// TwinCAT 3 PLC project TwinCAT_OpenFramework_Collections
// Title: TwinCAT Open Framework Collections
// Company: Oleksandr Tiutyk FOP
// Author: Oleksandr Tiutyk
// ProjectVersion: 1.0.13.0
// Description: Dynamic and static collections for TwinCAT.OpenFramework: ByteList, List, Dictionary, UniqueDataSet, Queue, Stack
// ProgramVersion: 3.1.4026.28
// libraries:
//   Tc2_Standard, * (Beckhoff Automation GmbH)
//   Tc2_System, * (Beckhoff Automation GmbH)
//   [TwinCAT Open Framework Core], * (Oleksandr Tiutyk FOP)
// project tree:
//   ByteList/ ByteList.TcPOU, ByteListEnumerator.TcPOU, IByteList.TcIO, IReadOnlyByteList.TcIO
//   Dictionary/ Dictionary.TcPOU, DictionaryEnumerator.TcPOU, IDictionary.TcIO, IReadOnlyDictionary.TcIO
//   / ICollection.TcIO
//   Internal/ CurrentNamespace.TcPOU, NamespaceExtractor.TcPOU
//   List/ IList.TcIO, IReadOnlyList.TcIO, List.TcPOU, ListEnumerator.TcPOU (not stored)
//   Queue/ IReadOnlyQueue.TcIO, IQueue.TcIO, Queue.TcPOU (not stored), QueueEnumerator.TcPOU
//   Stack/ IReadOnlyStack.TcIO, IStack.TcIO, Stack.TcPOU, StackEnumerator.TcPOU
//   UniqueDataSet/ UniqueDataSet.TcPOU, UniqueDataSetEnumerator.TcPOU, IUniqueDataSet.TcIO, IReadOnlyUniqueDataSet.TcIO
//   Version/ Global_Version.TcGVL
// (motion and I/O tree: see PLC project twincat_openframework_core)
// real-time tasks:
//   TASK PlcTask: cycle T#10ms, priority 20, ADS port 350
//   TASK TestTask: cycle T#10ms, priority 1, ADS port 351
//   TASK RunnerTestTask: cycle T#10ms, priority 2, ADS port 354
//   TASK HowToTask: cycle T#10ms, priority 22, ADS port 353
// variable links:

// ---- Version/Global_Version.TcGVL
{attribute 'TcGenerated'}
{attribute 'no-analysis'}
{attribute 'linkalways'}
// This function has been automatically generated from the project information.
VAR_GLOBAL CONSTANT
	{attribute 'const_non_replaced'}
	stLibVersion_TwinCAT_Open_Framework_Collections : ST_LibVersion := (iMajor := 1, iMinor := 0, iBuild := 13, iRevision := 0, nFlags := 0, sVersion := '1.0.13.0');
END_VAR

// ---- ByteList/IByteList.TcIO
(*
SPDX-FileCopyrightText: © 2026 Oleksandr Tiutyk <trofimich@gmail.com>
SPDX-License-Identifier: MIT
License: https://opensource.org/license/mit
*)

(*!
<summary>Provides byte sequence mutation and raw-memory copying.</summary>
<description>
Append adds bytes. LoadFrom writes at startIndex and sets Length to the end of the copied range, potentially
truncating the old tail. Input memory is borrowed for copying, never adopted. Remove by value is a no-op when
the value is absent, including on an empty collection. See method declarations for current safety limitations.
</description>
*)

INTERFACE IByteList EXTENDS IReadOnlyByteList

(*!
<summary>Appends the raw storage bytes of an ANY argument.</summary>
<description>
Borrows the argument for copying and uses its full runtime size, including string capacity and structure
padding. Not portable serialization or object cloning. Shares AppendData capacity checks, overlap support and
failure behavior.
</description>
*)
METHOD AppendAny : IByteList
VAR_INPUT
	data : ANY;
END_VAR
END_METHOD

(*!
<summary>Appends one byte by value.</summary>
<description>
Returns this list. Full static storage raises an exception; dynamic growth uses checked allocation and
terminal OOM handling.
</description>
*)
METHOD AppendByte : IByteList
VAR_INPUT
	value : BYTE;
END_VAR
END_METHOD

(*!
<summary>Appends bytes copied from a borrowed memory range.</summary>
<description>
Null data or zero dataSize is a no-op before size validation. Otherwise the source must be readable and
negative sizes or a resulting length outside DINT raise ArgumentOutOfRangeException before copying. Static
capacity exhaustion raises StaticCollectionFullException. Dynamic allocation uses checked growth and terminal
OOM handling. The existing growth increment (free capacity plus input size) is retained and must also fit. The
source may refer to this collection buffer, including overlapping ranges. The caller must provide a readable
range of dataSize bytes; growth keeps the old buffer alive until copying completes. No restriction to logical
Length is imposed on the source. Returns this list.
</description>
*)
METHOD AppendData : IByteList
VAR_INPUT
	data : POINTER TO BYTE;
	dataSize : TOF_Core.DINT_LENGTH;
END_VAR
END_METHOD

(*!
<summary>Appends the raw bytes referenced by a generic descriptor.</summary>
<description>
Borrows the descriptor without adopting or releasing it. Copies Address and Size without value conversion or
object cloning. Size above SignedInt32.MAX_VALUE raises ArgumentOutOfRangeException before narrowing,
including for a null Address. Shares AppendData aliasing and failure behavior.
</description>
*)
METHOD AppendGeneric : IByteList
VAR_INPUT
	data : TOF_Core.GENERIC_VALUE;
END_VAR
END_METHOD

(*!
<summary>Resets the byte count and optionally releases dynamic storage.</summary>
<description>
The default retains capacity for reuse. releaseDynamicMemory = TRUE deletes dynamic storage and sets capacity
to zero. Static storage is retained. Returns this list; old contents are no longer logical entries.
</description>
*)
METHOD Clear : IByteList
VAR_INPUT
	releaseDynamicMemory : BOOL := FALSE;
END_VAR
END_METHOD

(*!
<summary>Loads the full raw representation of an ANY argument at a position.</summary>
<description>
Delegates to LoadFromData using the runtime byte size, including padding and string capacity. Borrows the
source and may truncate the previous tail. Shares LoadFromData limits; not portable serialization.
</description>
*)
METHOD LoadFromAny : IByteList
VAR_INPUT
	data : ANY;
	startIndex : TOF_Core.DINT_INDEX := 0;
END_VAR
END_METHOD

(*!
<summary>Copies bytes at a position and sets Length to the end of the copy.</summary>
<description>
startIndex must lie between zero and old Length inclusive, and dataSize must be nonnegative; invalid arguments
raise ArgumentOutOfRangeException. Null data or zero size leaves Length unchanged after these checks. For a
nonempty copy, the resulting length is checked against DINT before arithmetic or mutation. The prefix remains
and the tail beyond the new end is logically truncated. Static capacity exhaustion raises
StaticCollectionFullException; dynamic growth uses checked allocation and terminal OOM handling. Internal
sources and overlapping ranges are supported. The caller must provide a readable source range of dataSize
bytes; the old buffer remains alive throughout copying on growth. No restriction to logical Length is imposed
on the source. Returns this list.
</description>
*)
METHOD LoadFromData : IByteList
VAR_INPUT
	data : POINTER TO BYTE;
	dataSize : TOF_Core.DINT_LENGTH;
	startIndex : TOF_Core.DINT_INDEX := 0;
END_VAR
END_METHOD

(*!
<summary>Loads the byte range referenced by a generic descriptor.</summary>
<description>
Borrows the descriptor without adoption or release. Size above SignedInt32.MAX_VALUE raises
ArgumentOutOfRangeException before narrowing, including for a null Address. Shares LoadFromData index checks,
truncation, aliasing and failure behavior.
</description>
*)
METHOD LoadFromGeneric : IByteList
VAR_INPUT
	data : TOF_Core.GENERIC_VALUE;
	startIndex : TOF_Core.DINT_INDEX := 0;
END_VAR
END_METHOD

(*!
<summary>Removes the first occurrence of a byte if present.</summary>
<description>
Removes only the first matching byte, compacts later bytes through RemoveAt and returns this list. An absent
value or an empty static or dynamic list leaves the collection unchanged without raising an exception for
absence. Capacity is retained. Requires an intact collection whose backing storage remains valid for its
logical contents.
</description>
*)
METHOD Remove : IByteList
VAR_INPUT
	value : BYTE;
END_VAR
END_METHOD

(*!
<summary>Removes a contiguous byte range and compacts remaining bytes.</summary>
<description>
Requires an existing index and a nonnegative count no greater than the remaining length; otherwise raises
ArgumentOutOfRangeException. The range is checked by subtraction before computing its end. Zero count is a
no-op only after index validation. Capacity is retained. Returns this list.
</description>
*)
METHOD RemoveAt : IByteList
VAR_INPUT
	index : TOF_Core.DINT_INDEX;
	count : TOF_Core.DINT_LENGTH := 1;
END_VAR
END_METHOD

(*!
<summary>Overwrites one existing byte.</summary>
<description>
Requires allocated storage and an index within Length; otherwise raises an exception. Length and Capacity are
unchanged. Returns this list.
</description>
*)
METHOD Set : IByteList
VAR_INPUT
	index : TOF_Core.DINT_INDEX;
	value : BYTE;
END_VAR
END_METHOD

END_INTERFACE

// ---- ByteList/IReadOnlyByteList.TcIO
(*
SPDX-FileCopyrightText: © 2026 Oleksandr Tiutyk <trofimich@gmail.com>
SPDX-License-Identifier: MIT
License: https://opensource.org/license/mit
*)

(*!
<summary>Provides indexed byte access and first-match searching.</summary>
<description>
Indices are zero-based. Get returns a byte value. Enumeration borrows the source, which must remain alive and
structurally unchanged during traversal.
</description>
*)

INTERFACE IReadOnlyByteList EXTENDS ICollection

(*!
<summary>Finds the first occurrence of a byte.</summary>
<description>
Searches from zero. TRUE makes index valid; on FALSE no index is promised. The collection is unchanged.
</description>
*)
METHOD Find : BOOL
VAR_INPUT
	value : BYTE;
END_VAR
VAR_OUTPUT
	index : TOF_Core.DINT_INDEX;
END_VAR
END_METHOD

(*!
<summary>Returns the byte at an existing zero-based position.</summary>
<description>
Raises an exception when backing storage is absent or the index is outside Length. The result is a byte copy.
</description>
*)
METHOD Get : BYTE
VAR_INPUT
	index : TOF_Core.DINT_INDEX;
END_VAR
END_METHOD

END_INTERFACE

// ---- Dictionary/IDictionary.TcIO
(*!
<summary>Associates generic keys with values.</summary>
<description>
SetGeneric retains an existing matching key and replaces its value. SetGeneric preserves disposal
responsibility when the same allocation is reused; transferred caller-side owning aliases must not be released
again. SetCopy prepares owned copies and cleans up prepared copies on failure before acceptance. Try
lookup/removal operations contain exceptions without rolling back partial effects. Generic query arguments are
borrowed by default. Explicitly requested release in Try operations is attempted even after lookup failure;
caller-side owning aliases are not reset. OBJECT keys are permitted when their descriptors refer to live
Object instances. A borrowed key (IsMemoryOwner = FALSE) is not owned or destroyed by the dictionary; its
owner must keep it alive for every operation that may access the stored key. An owned key must not be deleted
or transferred to another owner through a caller-side alias. While a key is stored, do not change data used by
the active comparison rules, its equality/hash results, or equality-relevant comparer configuration. Remove
the entry before such a change, then insert it again. Queries and callbacks must not mutate keys or reenter
collection mutation. Do not use explicit query release to dispose of a stored key or other storage still
retained by the collection. An address-based identity index must be rebuilt after address relocation; stale
indices must not be used. Borrowing does not pin an object or extend its lifetime. A copied object has its own
identity; lookup using the original requires an equality strategy under which original and copy are equal.
Default OBJECT lookup delegates to Object.Equals/GetHashCode; fields unrelated to equality/hash may change.
Discard and populate the index again after equality-relevant address relocation before further lookup. Lookup
uses one equality/hash strategy fixed for the collection lifetime; zero selects GENERIC_VALUE default equality
and hashing. A custom comparer is borrowed, stays alive and retains stable equality-relevant configuration.
Empty descriptors are supported unless rejected by a validator. No entry or enumeration order is guaranteed; a
position is a current storage slot, not a sorted rank. Do not modify stored descriptors through returned
references.
</description>
*)
(*
SPDX-FileCopyrightText: © 2026 Oleksandr Tiutyk <trofimich@gmail.com>
SPDX-License-Identifier: MIT
License: https://opensource.org/license/mit
*)

INTERFACE IDictionary EXTENDS IReadOnlyDictionary

(*!
<summary>Removes all entries and releases owned payload.</summary>
<description>
Disposal is best effort. Dynamic entry and index storage are released; static capacity and lifetime
comparer/validators are retained. References, positions and active enumeration are invalidated. Cleanup
callbacks must not reenter mutation.
</description>
*)
METHOD Clear : IDictionary
END_METHOD

(*!
<summary>Exposes the configured key validator.</summary>
<description>
Borrowed optional reference fixed at initialization. Zero means no validator. The collection does not own or
release it.
</description>
*)
{attribute 'monitoring' := 'call'}
PROPERTY FINAL KeyValidator : TOF_Core.IGenericValueValidator
GET
END_GET
END_PROPERTY

(*!
<summary>Removes the entry at a current storage position.</summary>
<description>
The index must be within Length and is not a sorted rank. Removal invalidates positions and references as
entries are compacted; owned payload disposal is best effort. Invalid indices raise an exception.
</description>
*)
METHOD RemoveAt : IDictionary
VAR_INPUT
	index : DINT;
END_VAR
END_METHOD

(*!
<summary>Copies source key and value storage and stores the prepared copies.</summary>
<description>
Original arguments remain borrowed. Object copies follow ICloneable; other payload is copied as bytes.
Prepared copies are released if copying or insertion fails before ownership is accepted. Exceptions propagate
after cleanup, without clearing terminal allocation state. The index output is meaningful only on success.
The original exception is captured before prepared-copy cleanup, so nested cleanup handling cannot replace
its payload. Terminal OOM takes precedence; capture failure still attempts prepared-copy disposal.
</description>
*)
//!<param name="key">Borrowed source key.</param>
//!<param name="value">Borrowed source value.</param>
//!<param name="keyIsObject">Explicitly interprets the key as object storage.</param>
//!<param name="valueIsObject">Explicitly interprets the value as object storage.</param>
METHOD SetCopy : IDictionary
VAR_INPUT
	key : ANY;
	value : ANY;
	keyIsObject : BOOL := FALSE;
	valueIsObject : BOOL := FALSE;
END_VAR
VAR_OUTPUT
	index : DINT;
END_VAR
END_METHOD

(*!
<summary>Stores a key-value pair, retaining the existing key when a matching entry is updated.</summary>
<description>
Uses the lifetime equality/hash strategy, with no ordering guarantee. Empty descriptors are permitted unless
rejected by a validator. A successful call accepts owned arguments; borrowed payload must remain alive while
stored. Validation, lookup and growth occur before acceptance; failure before acceptance leaves incoming
ownership with the caller. An unused owned incoming key and a displaced owned value are released after the new
entry is installed, unless their allocation is retained. Reusing the same allocation preserves existing
ownership or accepts incoming ownership; it never returns ownership implicitly. When key and value alias one
allocation, the key descriptor holds the pair's disposal responsibility. Input descriptor copies are not reset
in the caller: transferred owning aliases must not be released or reused as owners. Aliases must describe the
same allocation with compatible disposal semantics; overlapping owned ranges and ownership already held by
another entry or owner are not supported. Callbacks must not mutate or reenter this collection. Cleanup is
best effort through GENERIC_VALUE.Release and does not guarantee successful deallocation. The index output is
valid only on success.
</description>
*)
//!<param name="key">Incoming key descriptor; owned storage is transferred on success.</param>
//!<param name="value">Incoming value descriptor; owned storage is transferred on success.</param>
METHOD SetGeneric : IDictionary
VAR_INPUT
	key : TOF_Core.GENERIC_VALUE;
	value : TOF_Core.GENERIC_VALUE;
END_VAR
VAR_OUTPUT
	index : DINT;
END_VAR
END_METHOD

(*!
<summary>Attempts to remove a matching entry.</summary>
<description>
Returns the collection for chaining. removed is TRUE only after the matching entry has been removed; FALSE
means no completed removal was reported. Removal is not transactional and does not prove successful
destruction of an owned payload. Catches exceptions without propagating them or clearing terminal allocation
state. Partial changes are not rolled back. The query is borrowed by default. When releaseKey is explicitly
TRUE, attempts to release the supplied generic argument after lookup/removal even on failure. The caller must
have disposal rights and must not reuse aliases of an owned argument after release.
After nested calls and requested cleanup, a fatal allocation state forces the reported outcome to failure.
This does not roll back completed removal or reset the application-wide fatal latch.
</description>
*)
METHOD TryRemoveByGenericKey : IDictionary
VAR_INPUT
	key : TOF_Core.GENERIC_VALUE;
	releaseKey : BOOL := FALSE;
END_VAR
VAR_OUTPUT
	removed : BOOL;
END_VAR
END_METHOD

(*!
<summary>Attempts to remove a matching entry.</summary>
<description>
Returns the collection for chaining. removed is TRUE only after the matching entry has been removed; FALSE
means no completed removal was reported. Removal is not transactional and does not prove successful
destruction of an owned payload. Catches exceptions without propagating them or clearing terminal allocation
state. Partial changes are not rolled back. The raw ANY argument is borrowed without cloning or ownership
transfer. keyIsObject = TRUE requires a live Object function-block instance, not a pointer or interface
variable. FALSE uses ordinary runtime type mapping. The caller keeps the query storage alive for the call.
After nested calls and requested cleanup, a fatal allocation state forces the reported outcome to failure.
This does not roll back completed removal or reset the application-wide fatal latch.
</description>
*)
//!<param name="keyIsObject">Explicitly interprets the raw argument as a live Object instance.</param>
METHOD TryRemoveByKey : IDictionary
VAR_INPUT
	key : ANY;
	keyIsObject : BOOL := FALSE;
END_VAR
VAR_OUTPUT
	removed : BOOL;
END_VAR
END_METHOD

(*!
<summary>Exposes the configured value validator.</summary>
<description>
Borrowed optional reference fixed at initialization. Zero means no validator. The collection does not own or
release it.
</description>
*)
{attribute 'monitoring' := 'call'}
PROPERTY FINAL ValueValidator : TOF_Core.IGenericValueValidator
GET
END_GET
END_PROPERTY

END_INTERFACE

// ---- Dictionary/IReadOnlyDictionary.TcIO
(*!
<summary>Associates generic keys with values.</summary>
<description>
Try lookup/removal operations contain exceptions without rolling back partial effects. Generic query arguments
are borrowed by default. Explicitly requested release in Try operations is attempted even after lookup
failure; caller-side owning aliases are not reset. OBJECT keys are permitted when their descriptors refer to
live Object instances. A borrowed key (IsMemoryOwner = FALSE) is not owned or destroyed by the dictionary; its
owner must keep it alive for every operation that may access the stored key. An owned key must not be deleted
or transferred to another owner through a caller-side alias. While a key is stored, do not change data used by
the active comparison rules, its equality/hash results, or equality-relevant comparer configuration. Remove
the entry before such a change, then insert it again. Queries and callbacks must not mutate keys or reenter
collection mutation. Do not use explicit query release to dispose of a stored key or other storage still
retained by the collection. An address-based identity index must be rebuilt after address relocation; stale
indices must not be used. Borrowing does not pin an object or extend its lifetime. A copied object has its own
identity; lookup using the original requires an equality strategy under which original and copy are equal.
Default OBJECT lookup delegates to Object.Equals/GetHashCode; fields unrelated to equality/hash may change.
Discard and populate the index again after equality-relevant address relocation before further lookup. Lookup
uses one equality/hash strategy fixed for the collection lifetime; zero selects GENERIC_VALUE default equality
and hashing. A custom comparer is borrowed, stays alive and retains stable equality-relevant configuration.
Empty descriptors are supported unless rejected by a validator. No entry or enumeration order is guaranteed; a
position is a current storage slot, not a sorted rank. Do not modify stored descriptors through returned
references.
</description>
*)
(*
SPDX-FileCopyrightText: © 2026 Oleksandr Tiutyk <trofimich@gmail.com>
SPDX-License-Identifier: MIT
License: https://opensource.org/license/mit
*)

INTERFACE IReadOnlyDictionary EXTENDS ICollection

(*!
<summary>Reports whether a matching entry exists for a borrowed generic query.</summary>
<description>
The query is borrowed by default. Explicit release requests disposal of owned query storage after lookup
completes, including a missing result. Requested release is attempted after both successful lookup and lookup
failure. Before cleanup, the original framework exception is retained and a borrowed static system exception
is cloned to preserve its code, catch point and timestamps across cleanup callbacks. The captured exception is
then propagated through ExceptionManager.Throw in the current cyclic task; native errors use the framework
SystemException representation. If capturing the system exception fails with terminal OOM, query cleanup is
still attempted and terminal OOM takes precedence. Terminal allocation state is never cleared. Release is best
effort and does not prove successful deallocation. Cleanup callbacks must not reenter collection mutation.
Release resets only the local descriptor copy; the caller must have disposal rights and must not reuse or
release owning aliases afterwards. Borrowed payload is not freed.
</description>
*)
METHOD ContainsGenericKey : BOOL
VAR_INPUT
	key : TOF_Core.GENERIC_VALUE;
	releaseKey : BOOL := FALSE;
END_VAR
END_METHOD

(*!
<summary>Reports whether a matching raw query exists.</summary>
<description>
The raw ANY argument is borrowed without cloning or ownership transfer. keyIsObject = TRUE requires a live
Object function-block instance, not a pointer or interface variable. FALSE uses ordinary runtime type mapping.
The caller keeps the query storage alive for the call.
</description>
*)
//!<param name="keyIsObject">Explicitly interprets the raw argument as a live Object instance.</param>
METHOD ContainsKey : BOOL
VAR_INPUT
	key : ANY;
	keyIsObject : BOOL := FALSE;
END_VAR
END_METHOD

(*!
<summary>Returns the matching entry position, or a negative value when absent.</summary>
<description>
The query is borrowed by default. Explicit release requests disposal of owned query storage after lookup
completes, including a missing result. Requested release is attempted after both successful lookup and lookup
failure. Before cleanup, the original framework exception is retained and a borrowed static system exception
is cloned to preserve its code, catch point and timestamps across cleanup callbacks. The captured exception is
then propagated through ExceptionManager.Throw in the current cyclic task; native errors use the framework
SystemException representation. If capturing the system exception fails with terminal OOM, query cleanup is
still attempted and terminal OOM takes precedence. Terminal allocation state is never cleared. Release is best
effort and does not prove successful deallocation. Cleanup callbacks must not reenter collection mutation.
Release resets only the local descriptor copy; the caller must have disposal rights and must not reuse or
release owning aliases afterwards. Borrowed payload is not freed. The position is a current storage slot with
no sorted-rank guarantee; mutation may invalidate it.
</description>
*)
METHOD GetGenericKeyPosition : DINT
VAR_INPUT
	key : TOF_Core.GENERIC_VALUE;
	releaseKey : BOOL := FALSE;
END_VAR
END_METHOD

(*!
<summary>Returns the matching storage position, or a negative value when absent.</summary>
<description>
The raw ANY argument is borrowed without cloning or ownership transfer. keyIsObject = TRUE requires a live
Object function-block instance, not a pointer or interface variable. FALSE uses ordinary runtime type mapping.
The caller keeps the query storage alive for the call. The position is a current storage slot with no
sorted-rank guarantee; mutation may invalidate it.
</description>
*)
//!<param name="keyIsObject">Explicitly interprets the raw argument as a live Object instance.</param>
METHOD GetKeyPosition : DINT
VAR_INPUT
	key : ANY;
	keyIsObject : BOOL := FALSE;
END_VAR
END_METHOD

(*!
<summary>Borrows the entry at a current storage position.</summary>
<description>
The index must be within Length and is not a sorted rank; otherwise an exception is raised. The returned
descriptor reference and payload remain collection-owned or borrowed from their original owner. Do not mutate
the descriptor or dispose of its payload through this view. Mutation or destruction may invalidate the
reference.
</description>
*)
METHOD GetKeyValuePairByIndex : REFERENCE TO TOF_Core.GENERIC_KEY_VALUE_PAIR
VAR_INPUT
	index : DINT;
END_VAR
END_METHOD

(*!
<summary>Attempts to find a value by its key.</summary>
<description>
Returns TRUE when a value is found. Use the output only on TRUE; no payload is cloned. Catches exceptions
without propagating them or clearing terminal allocation state. Partial changes are not rolled back. The query
is borrowed by default. When releaseKey is explicitly TRUE, attempts to release the supplied generic argument
after lookup/removal even on failure. The caller must have disposal rights and must not reuse aliases of an
owned argument after release. A successful output is a borrowed descriptor copy; IsMemoryOwner does not
transfer disposal rights to the caller. Stored payload must not be released through the output.
After nested calls and requested cleanup, a fatal allocation state forces the reported outcome to failure.
This does not roll back completed removal or reset the application-wide fatal latch.
</description>
*)
METHOD TryGetValueByGenericKey : BOOL
VAR_INPUT
	key : TOF_Core.GENERIC_VALUE;
	releaseKey : BOOL := FALSE;
END_VAR
VAR_OUTPUT
	value : TOF_Core.GENERIC_VALUE;
END_VAR
END_METHOD

(*!
<summary>Attempts to find a value by its key.</summary>
<description>
Returns TRUE when a value is found. Use the output only on TRUE; no payload is cloned. Catches exceptions
without propagating them or clearing terminal allocation state. Partial changes are not rolled back. The raw
ANY argument is borrowed without cloning or ownership transfer. keyIsObject = TRUE requires a live Object
function-block instance, not a pointer or interface variable. FALSE uses ordinary runtime type mapping. The
caller keeps the query storage alive for the call. A successful output is a borrowed descriptor copy;
IsMemoryOwner does not transfer disposal rights to the caller. Stored payload must not be released through the
output.
After nested calls and requested cleanup, a fatal allocation state forces the reported outcome to failure.
This does not roll back completed removal or reset the application-wide fatal latch.
</description>
*)
//!<param name="keyIsObject">Explicitly interprets the raw argument as a live Object instance.</param>
METHOD TryGetValueByKey : BOOL
VAR_INPUT
	key : ANY;
	keyIsObject : BOOL := FALSE;
END_VAR
VAR_OUTPUT
	value : TOF_Core.GENERIC_VALUE;
END_VAR
END_METHOD

END_INTERFACE

// ---- ICollection.TcIO
(*
SPDX-FileCopyrightText: © 2026 Oleksandr Tiutyk <trofimich@gmail.com>
SPDX-License-Identifier: MIT
License: https://opensource.org/license/mit
*)

(*!
<summary>Provides collection size, capacity and enumeration.</summary>
<description>
Does not transfer ownership of the collection. CreateEnumerator follows IEnumerable: the caller owns the
dynamic cursor and keeps the source alive. Full describes fixed-capacity exhaustion, not heap availability. No
synchronization or snapshot guarantee is supplied by this interface.
</description>
*)

INTERFACE ICollection EXTENDS TOF_Core.IEnumerable

(*!
<summary>Reports the currently allocated number of slots.</summary>
<description>
Units are bytes for ByteList and entries for other collections. Static capacity is fixed; dynamic capacity can
change on growth or clearing. This is not a guarantee that the next allocation succeeds.
</description>
*)
{attribute 'monitoring' := 'call'}
PROPERTY Capacity : TOF_Core.DINT_LENGTH
GET
END_GET
END_PROPERTY

(*!
<summary>Reports whether storage can grow dynamically.</summary>
<description>
Static capacity zero selects dynamic storage. Dynamic collections can still fail to allocate.
</description>
*)
{attribute 'monitoring' := 'call'}
PROPERTY Dynamic : BOOL
GET
END_GET
END_PROPERTY

(*!
<summary>Reports whether the collection has no entries.</summary>
<description>
Reflects Length; not a check of payload lifetime or memory health.
</description>
*)
{attribute 'monitoring' := 'call'}
PROPERTY Empty : BOOL
GET
END_GET
END_PROPERTY

(*!
<summary>Reports whether fixed-capacity storage has no free slot.</summary>
<description>
Dynamic collections report FALSE even when Length equals Capacity. This does not guarantee available heap
memory.
</description>
*)
{attribute 'monitoring' := 'call'}
PROPERTY Full : BOOL
GET
END_GET
END_PROPERTY

(*!
<summary>Reports the number of stored entries.</summary>
<description>
Units are bytes for ByteList and entries for other collections. Existing positions range from zero through
Length minus one.
</description>
*)
{attribute 'OPC.UA.DA.Property' := '1'}
{attribute 'monitoring' := 'call'}
PROPERTY Length : TOF_Core.DINT_LENGTH
GET
END_GET
END_PROPERTY

END_INTERFACE

// ---- List/IList.TcIO
(*
SPDX-FileCopyrightText: © 2026 Oleksandr Tiutyk <trofimich@gmail.com>
SPDX-License-Identifier: MIT
License: https://opensource.org/license/mit
*)

(*!
<summary>Provides generic-value insertion, replacement, removal and in-place reordering.</summary>
<description>
Successful insertion transfers disposal responsibility for owned payload; borrowed payload must remain alive
while stored. The caller-side descriptor copy is not reset and must not be released again after transfer.
Independent owning aliases and overlapping owned allocations are unsupported. Get and FindSingle do not
transfer ownership back. Removal releases owned payload. Validators are borrowed. Sort and Swap change entry
order without changing collection length or payload ownership. Same-allocation replacement preserves
collection ownership; aliases must have compatible disposal semantics.
</description>
*)

INTERFACE IList EXTENDS IReadOnlyList

(*!
<summary>Copies a value and appends the owned descriptor.</summary>
<description>
Borrows the original during the call. isObject = TRUE requires a live Object FB instance implementing
ICloneable; other data is copied as bytes without recursively cloning references. A prepared copy is released
if insertion fails before acceptance; exceptions propagate. Engine-managed exception objects are unsupported.
index is meaningful only on success.
The original exception is captured before prepared-copy cleanup, so nested cleanup handling cannot replace
its payload. Terminal OOM takes precedence; capture failure still attempts prepared-copy disposal.
</description>
*)
METHOD AppendCopy : IList
VAR_INPUT
	value : ANY;
	isObject : BOOL := FALSE;
END_VAR
VAR_OUTPUT
	index : TOF_Core.DINT_INDEX;
END_VAR
END_METHOD

(*!
<summary>Appends a descriptor to the list.</summary>
<description>
Successful insertion transfers disposal responsibility for owned payload; borrowed payload must remain alive
while stored. The caller-side descriptor copy is not reset and must not be released again after transfer.
Independent owning aliases and overlapping owned allocations are unsupported. Delegates to InsertGeneric;
index is meaningful only on success.
</description>
*)
METHOD AppendGeneric : IList
VAR_INPUT
	value : TOF_Core.GENERIC_VALUE;
END_VAR
VAR_OUTPUT
	index : TOF_Core.DINT_INDEX;
END_VAR
END_METHOD

(*!
<summary>Removes all entries and releases dynamic backing storage.</summary>
<description>
Owned payload is released best effort through GENERIC_VALUE.Release; borrowed storage is not freed. Static
capacity and the borrowed validator are retained. Dynamic capacity becomes zero. Returns this collection and
invalidates positions and views. Cleanup callbacks must not reenter mutation.
</description>
*)
METHOD Clear : IList
END_METHOD

(*!
<summary>Reports whether storage can grow dynamically.</summary>
<description>
Static capacity zero selects dynamic storage. Dynamic collections can still fail to allocate.
</description>
*)
{attribute 'monitoring' := 'call'}
PROPERTY Dynamic : BOOL
GET
END_GET
END_PROPERTY

(*!
<summary>Copies a value and inserts it at the requested position.</summary>
<description>
Borrows the original during the call. isObject = TRUE requires a live Object FB instance implementing
ICloneable; other data is copied as bytes without recursively cloning references. A prepared copy is released
if insertion fails before acceptance; exceptions propagate. Engine-managed exception objects are unsupported.
The position may range from zero through Length inclusive.
The original exception is captured before prepared-copy cleanup, so nested cleanup handling cannot replace
its payload. Terminal OOM takes precedence; capture failure still attempts prepared-copy disposal.
</description>
*)
METHOD InsertCopy : IList
VAR_INPUT
	index : TOF_Core.DINT_INDEX;
	value : ANY;
	isObject : BOOL := FALSE;
END_VAR
END_METHOD

(*!
<summary>Inserts a descriptor and shifts subsequent entries to the right.</summary>
<description>
Successful insertion transfers disposal responsibility for owned payload; borrowed payload must remain alive
while stored. The caller-side descriptor copy is not reset and must not be released again after transfer.
Independent owning aliases and overlapping owned allocations are unsupported. index may range from zero
through Length inclusive. Invalid indices and full static storage raise exceptions. Validation precedes
insertion. Dynamic growth rejects nonpositive increments and unrepresentable capacity or allocation sizes
before insertion.
</description>
*)
METHOD InsertGeneric : IList
VAR_INPUT
	index : TOF_Core.DINT_INDEX;
	value : TOF_Core.GENERIC_VALUE;	
END_VAR
END_METHOD

(*!
<summary>Removes an existing list entry and compacts subsequent entries.</summary>
<description>
Invalid indices raise an exception. Owned payload is released best effort through GENERIC_VALUE.Release;
borrowed payload is not freed. Returns this list. Positions and descriptor references may change; cleanup
callbacks must not reenter mutation.
</description>
*)
METHOD RemoveAt : IList
VAR_INPUT
	index : TOF_Core.DINT_INDEX;
END_VAR
END_METHOD

(*!
<summary>Removes the first list entry equal to a borrowed query.</summary>
<description>
Uses default GENERIC_VALUE equality; isObject = TRUE requires a live Object FB instance. Reports removed on a
successful match and returns this list. Owned stored payload is released; the query is not adopted or
separately released. Equality exceptions propagate.
</description>
*)
METHOD RemoveFirst : IList
VAR_INPUT
	value : ANY;
	isObject : BOOL := FALSE;
END_VAR
VAR_OUTPUT
	removed : BOOL;
END_VAR
END_METHOD

(*!
<summary>Removes predicate matches while traversing from the end.</summary>
<description>
skip counts matches from the end. A null predicate or maxRemoved = 0 performs no removal. Removes at most
maxRemoved matching entries after skipping the requested matches. Stops immediately after reaching the limit,
without invoking the predicate for remaining entries. Predicate exceptions propagate after any completed
removals, without rollback. removedCount counts completed removals. Callbacks must not mutate the traversed
collection.
</description>
*)
METHOD RemoveMatched : IList
VAR_INPUT
	predicate : TOF_Core.IPredicate;
	skip : UDINT := 0;
	maxRemoved : UDINT := TOF_Core.UnsignedInt32.MAX_VALUE;
END_VAR
VAR_OUTPUT
	removedCount : DINT;
END_VAR
END_METHOD

(*!
<summary>Copies a value and stores it through SetGeneric.</summary>
<description>
Borrows the original during the call. isObject = TRUE requires a live Object FB instance implementing
ICloneable; other data is copied as bytes without recursively cloning references. A prepared copy is released
if insertion fails before acceptance; exceptions propagate. Engine-managed exception objects are unsupported.
Any index output is meaningful only on success.
The original exception is captured before prepared-copy cleanup, so nested cleanup handling cannot replace
its payload. Terminal OOM takes precedence; capture failure still attempts prepared-copy disposal.
</description>
*)
METHOD SetCopy : IList
VAR_INPUT
	index : TOF_Core.DINT_INDEX;
	value : ANY;
	isObject : BOOL := FALSE;
END_VAR
END_METHOD

(*!
<summary>Replaces the descriptor at an existing list position.</summary>
<description>
Successful replacement transfers disposal responsibility for owned payload; borrowed payload must remain alive
while stored. The caller-side descriptor copy is not reset and must not be released again after transfer.
Invalid indices and rejected validation raise exceptions before replacement. Reusing the same allocation
preserves existing ownership or accepts incoming ownership without releasing that allocation. Aliases must
have compatible disposal semantics; independently owned aliases and overlapping owned ranges are unsupported.
A different displaced allocation is released best effort after installing the new descriptor. Cleanup
callbacks must not reenter collection mutation.
</description>
*)
METHOD SetGeneric : IList
VAR_INPUT
	index : TOF_Core.DINT_INDEX;
	value : TOF_Core.GENERIC_VALUE;	
END_VAR
END_METHOD

(*!
<summary>Reorders list entries according to a generic-value comparer.</summary>
<description>
An omitted or null comparer selects GENERIC_VALUE.CompareTo. An explicit comparer takes precedence and must
provide a consistent order for the borrowed stored values. The default order follows Core numeric, text,
temporal and OBJECT rules; incompatible pairs raise GenericConversionNotSupportedException and OBJECT needs
IComparable. Empty/single lists return without comparing. Callbacks must not mutate operands or the list.
Comparison failure may leave entries partially reordered; all descriptors and payload ownership are retained.
</description>
*)
//!<param name="comparer">Optional borrowed ordering strategy; zero selects GENERIC_VALUE.CompareTo.</param>
//!<param name="direction">Requested ordering direction.</param>
METHOD Sort : IList
VAR_INPUT
	comparer : TOF_Core.IComparer := 0;
	direction : TOF_Core.SORT_DIRECTION := TOF_Core.SORT_DIRECTION.ASCENDING;
END_VAR
END_METHOD

(*!
<summary>Exchanges two positions without cloning or releasing payload.</summary>
<description>
Returns this list. Different indices must be valid or an exception is raised. Current implementation returns
immediately for equal indices without validating them. Payload ownership is preserved.
</description>
*)
METHOD Swap : IList
VAR_INPUT
	index1 : TOF_Core.DINT_INDEX;
	index2 : TOF_Core.DINT_INDEX;
END_VAR
END_METHOD

(*!
<summary>Exposes the configured value validator.</summary>
<description>
Borrowed optional reference fixed at initialization. Zero means no validator. The collection does not own or
release it.
</description>
*)
{attribute 'monitoring' := 'call'}
PROPERTY ValueValidator : TOF_Core.IGenericValueValidator
GET
END_GET
END_PROPERTY

END_INTERFACE

// ---- List/IReadOnlyList.TcIO
(*
SPDX-FileCopyrightText: © 2026 Oleksandr Tiutyk <trofimich@gmail.com>
SPDX-License-Identifier: MIT
License: https://opensource.org/license/mit
*)

(*!
<summary>Provides indexed access and searching without operations that change list entries or their order.</summary>
<description>
This interface does not expose insertion, removal, replacement or reordering. It is a view, not an immutable
snapshot: changes through another mutable reference can invalidate positions. Borrowed descriptors and payload
require the source collection to remain alive. ContainsGeneric currently defaults to releasing an owned query.
Get and FindSingle return borrowed views even when their descriptor carries IsMemoryOwner; a descriptor copy
does not transfer ownership.
</description>
*)
INTERFACE IReadOnlyList EXTENDS ICollection

(*!
<summary>Searches for a value using default generic equality.</summary>
<description>
Borrows the ANY argument during a linear search without cloning or releasing it. isObject = TRUE means a live
Object FB instance, not a pointer or interface variable. Equality exceptions propagate; callbacks that mutate
the collection can invalidate traversal.
</description>
*)
METHOD Contains : BOOL
VAR_INPUT
	value : ANY;
	isObject : BOOL := FALSE;
END_VAR
END_METHOD

(*!
<summary>Searches for an equal generic value and optionally releases the query.</summary>
<description>
Uses GENERIC_VALUE.Equals in a linear search. releaseValue defaults to TRUE: after a completed search, Release
is called on the local query copy, including on a miss. Caller-side aliases are not reset. The query must not
own storage retained by the collection. Requested release is attempted after both successful lookup and lookup
failure. Before cleanup, the original framework exception is retained and a borrowed static system exception
is cloned to preserve its code, catch point and timestamps across cleanup callbacks. The captured exception is
then propagated through ExceptionManager.Throw in the current cyclic task; native errors use the framework
SystemException representation. If capturing the system exception fails with terminal OOM, query cleanup is
still attempted and terminal OOM takes precedence. Terminal allocation state is never cleared. Release is best
effort and does not prove successful deallocation. Cleanup callbacks must not reenter collection mutation.
</description>
*)
METHOD ContainsGeneric : BOOL
VAR_INPUT
	value : TOF_Core.GENERIC_VALUE;
	releaseValue : BOOL := TRUE;
END_VAR
END_METHOD

(*!
<summary>Finds a predicate match in the requested traversal direction.</summary>
<description>
skip counts matches, not visited entries. A null predicate or no match returns FALSE; outputs are meaningful
only on TRUE. The result is borrowed even if IsMemoryOwner is TRUE. Predicate input uses AsAnyType without
preserving the explicit generic OBJECT category. Predicate exceptions propagate; callbacks must not mutate the
traversed collection.
</description>
*)
METHOD FindSingle : BOOL
VAR_INPUT
	predicate : TOF_Core.IPredicate;
	skip : UDINT := 0;
	searchDirection : TOF_Core.SEARCH_DIRECTION := TOF_Core.SEARCH_DIRECTION.FROM_BEGINNING;
END_VAR
VAR_OUTPUT
	value : TOF_Core.GENERIC_VALUE;
	index : TOF_Core.DINT_INDEX;
END_VAR
END_METHOD

(*!
<summary>Reports whether fixed-capacity storage has no free slot.</summary>
<description>
Dynamic collections report FALSE even when Length equals Capacity. This does not guarantee available heap
memory.
</description>
*)
{attribute 'monitoring' := 'call'}
PROPERTY FINAL Full : BOOL
GET
END_GET
END_PROPERTY

(*!
<summary>Borrows the descriptor at a zero-based list position.</summary>
<description>
An out-of-range index raises an exception. Returned descriptors and payload are borrowed, not clones. Do not
modify descriptor metadata or release payload through this view, even when IsMemoryOwner is TRUE. Keep the
source and borrowed storage alive; mutation or destruction can invalidate the view.
</description>
*)
METHOD Get : REFERENCE TO TOF_Core.GENERIC_VALUE
VAR_INPUT
	index : TOF_Core.DINT_INDEX;
END_VAR
END_METHOD

END_INTERFACE

// ---- Queue/IReadOnlyQueue.TcIO
(*
SPDX-FileCopyrightText: © 2026 Oleksandr Tiutyk <trofimich@gmail.com>
SPDX-License-Identifier: MIT
License: https://opensource.org/license/mit
*)

(*!
<summary>Provides FIFO head inspection, indexed access and membership queries.</summary>
<description>
Returned descriptors and payload are borrowed, not clones. Do not modify descriptor metadata or release
payload through this view, even when IsMemoryOwner is TRUE. Keep the source and borrowed storage alive;
mutation or destruction can invalidate the view. ContainsGeneric currently defaults to releasing an owned
query.
</description>
*)

INTERFACE IReadOnlyQueue EXTENDS ICollection

(*!
<summary>Searches for a value using default generic equality.</summary>
<description>
Borrows the ANY argument during a linear search without cloning or releasing it. isObject = TRUE means a live
Object FB instance, not a pointer or interface variable. Equality exceptions propagate; callbacks that mutate
the collection can invalidate traversal.
</description>
*)
METHOD Contains : BOOL
VAR_INPUT
	value : ANY;
	isObject : BOOL := FALSE;
END_VAR
END_METHOD

(*!
<summary>Searches for an equal generic value and optionally releases the query.</summary>
<description>
Uses GENERIC_VALUE.Equals in a linear search. releaseValue defaults to TRUE: after a completed search, Release
is called on the local query copy, including on a miss. Caller-side aliases are not reset. The query must not
own storage retained by the collection. Requested release is attempted after both successful lookup and lookup
failure. Before cleanup, the original framework exception is retained and a borrowed static system exception
is cloned to preserve its code, catch point and timestamps across cleanup callbacks. The captured exception is
then propagated through ExceptionManager.Throw in the current cyclic task; native errors use the framework
SystemException representation. If capturing the system exception fails with terminal OOM, query cleanup is
still attempted and terminal OOM takes precedence. Terminal allocation state is never cleared. Release is best
effort and does not prove successful deallocation. Cleanup callbacks must not reenter collection mutation.
</description>
*)
METHOD ContainsGeneric : BOOL
VAR_INPUT
	value : TOF_Core.GENERIC_VALUE;
	releaseValue : BOOL := TRUE;
END_VAR
END_METHOD

(*!
<summary>Borrows the descriptor at a zero-based queue position.</summary>
<description>
Position zero is the head. An out-of-range index raises an exception. Returned descriptors and payload are
borrowed, not clones. Do not modify descriptor metadata or release payload through this view, even when
IsMemoryOwner is TRUE. Keep the source and borrowed storage alive; mutation or destruction can invalidate the
view.
</description>
*)
METHOD GetByIndex : REFERENCE TO TOF_Core.GENERIC_VALUE
VAR_INPUT
	index : TOF_Core.DINT_INDEX;
END_VAR
END_METHOD

(*!
<summary>Borrows the FIFO head without removing it.</summary>
<description>
An empty queue raises CollectionEmptyException. Returned descriptors and payload are borrowed, not clones. Do
not modify descriptor metadata or release payload through this view, even when IsMemoryOwner is TRUE. Keep the
source and borrowed storage alive; mutation or destruction can invalidate the view.
</description>
*)
METHOD Peek : REFERENCE TO TOF_Core.GENERIC_VALUE
END_METHOD

END_INTERFACE

// ---- Queue/IQueue.TcIO
(*
SPDX-FileCopyrightText: © 2026 Oleksandr Tiutyk <trofimich@gmail.com>
SPDX-License-Identifier: MIT
License: https://opensource.org/license/mit
*)

(*!
<summary>Provides FIFO insertion and destructive head removal.</summary>
<description>
Successful insertion transfers disposal responsibility for owned payload; borrowed payload must remain alive
while stored. The caller-side descriptor copy is not reset and must not be released again after transfer.
Independent owning aliases and overlapping owned allocations are unsupported. Peek borrows the head;
RemoveFirst releases it rather than transferring it to the caller. Clear releases owned payload and dynamic
backing storage.
</description>
*)

INTERFACE IQueue EXTENDS IReadOnlyQueue

(*!
<summary>Removes all entries and releases dynamic backing storage.</summary>
<description>
Owned payload is released best effort through GENERIC_VALUE.Release; borrowed storage is not freed. Static
capacity and the borrowed validator are retained. Dynamic capacity becomes zero. Returns this collection and
invalidates positions and views. Cleanup callbacks must not reenter mutation.
</description>
*)
METHOD Clear : IQueue
END_METHOD

(*!
<summary>Copies a value and appends it to the FIFO tail.</summary>
<description>
Borrows the original during the call. isObject = TRUE requires a live Object FB instance implementing
ICloneable; other data is copied as bytes without recursively cloning references. A prepared copy is released
if insertion fails before acceptance; exceptions propagate. Engine-managed exception objects are unsupported.
The original exception is captured before prepared-copy cleanup, so nested cleanup handling cannot replace
its payload. Terminal OOM takes precedence; capture failure still attempts prepared-copy disposal.
</description>
*)
METHOD EnqueueCopy : IQueue
VAR_INPUT
	value : ANY;
	isObject : BOOL := FALSE;
END_VAR
END_METHOD

(*!
<summary>Appends a descriptor after the FIFO tail.</summary>
<description>
Successful insertion transfers disposal responsibility for owned payload; borrowed payload must remain alive
while stored. The caller-side descriptor copy is not reset and must not be released again after transfer.
Independent owning aliases and overlapping owned allocations are unsupported. Full static storage raises an
exception. A configured validator is invoked once before any capacity growth or ownership acceptance.
Validation failure leaves the buffer, Length and incoming ownership unchanged; its exception propagates.
Validator callbacks must not mutate this collection.
</description>
*)
METHOD EnqueueGeneric : IQueue
VAR_INPUT
	value : TOF_Core.GENERIC_VALUE;
END_VAR
END_METHOD

(*!
<summary>Removes the FIFO head without transferring it to the caller.</summary>
<description>
An empty queue raises CollectionEmptyException. Owned head storage is released best effort, not returned to
the caller. Remaining descriptors shift left in linear time. Returns this queue; positions and views may
change. Cleanup callbacks must not reenter mutation.
</description>
*)
METHOD RemoveFirst : IQueue
END_METHOD

(*!
<summary>Exposes the configured value validator.</summary>
<description>
Borrowed optional reference fixed at initialization. Zero means no validator. The collection does not own or
release it.
</description>
*)
{attribute 'monitoring' := 'call'}
PROPERTY ValueValidator : TOF_Core.IGenericValueValidator
GET
END_GET
END_PROPERTY

END_INTERFACE

// ---- Stack/IReadOnlyStack.TcIO
(*
SPDX-FileCopyrightText: © 2026 Oleksandr Tiutyk <trofimich@gmail.com>
SPDX-License-Identifier: MIT
License: https://opensource.org/license/mit
*)

(*!
<summary>Provides LIFO top inspection, indexed access and membership queries.</summary>
<description>
Returned descriptors and payload are borrowed, not clones. Do not modify descriptor metadata or release
payload through this view, even when IsMemoryOwner is TRUE. Keep the source and borrowed storage alive;
mutation or destruction can invalidate the view. ContainsGeneric currently defaults to releasing an owned
query.
</description>
*)

INTERFACE IReadOnlyStack EXTENDS ICollection

(*!
<summary>Searches for a value using default generic equality.</summary>
<description>
Borrows the ANY argument during a linear search without cloning or releasing it. isObject = TRUE means a live
Object FB instance, not a pointer or interface variable. Equality exceptions propagate; callbacks that mutate
the collection can invalidate traversal.
</description>
*)
METHOD Contains : BOOL
VAR_INPUT
	value : ANY;
	isObject : BOOL := FALSE;
END_VAR
END_METHOD

(*!
<summary>Searches for an equal generic value and optionally releases the query.</summary>
<description>
Uses GENERIC_VALUE.Equals in a linear search. releaseValue defaults to TRUE: after a completed search, Release
is called on the local query copy, including on a miss. Caller-side aliases are not reset. The query must not
own storage retained by the collection. Requested release is attempted after both successful lookup and lookup
failure. Before cleanup, the original framework exception is retained and a borrowed static system exception
is cloned to preserve its code, catch point and timestamps across cleanup callbacks. The captured exception is
then propagated through ExceptionManager.Throw in the current cyclic task; native errors use the framework
SystemException representation. If capturing the system exception fails with terminal OOM, query cleanup is
still attempted and terminal OOM takes precedence. Terminal allocation state is never cleared. Release is best
effort and does not prove successful deallocation. Cleanup callbacks must not reenter collection mutation.
</description>
*)
METHOD ContainsGeneric : BOOL
VAR_INPUT
	value : TOF_Core.GENERIC_VALUE;
	releaseValue : BOOL := TRUE;
END_VAR
END_METHOD

(*!
<summary>Borrows the descriptor at a zero-based stack position.</summary>
<description>
Position zero is the top; increasing indices move toward the bottom. An out-of-range index raises an
exception. Returned descriptors and payload are borrowed, not clones. Do not modify descriptor metadata or
release payload through this view, even when IsMemoryOwner is TRUE. Keep the source and borrowed storage
alive; mutation or destruction can invalidate the view.
</description>
*)
METHOD GetByIndex : REFERENCE TO TOF_Core.GENERIC_VALUE
VAR_INPUT
	index : TOF_Core.DINT_INDEX;
END_VAR
END_METHOD

(*!
<summary>Borrows the LIFO top without removing it.</summary>
<description>
An empty stack raises CollectionEmptyException. Returned descriptors and payload are borrowed, not clones. Do
not modify descriptor metadata or release payload through this view, even when IsMemoryOwner is TRUE. Keep the
source and borrowed storage alive; mutation or destruction can invalidate the view.
</description>
*)
METHOD Peek : REFERENCE TO TOF_Core.GENERIC_VALUE
END_METHOD

END_INTERFACE

// ---- Stack/IStack.TcIO
(*
SPDX-FileCopyrightText: © 2026 Oleksandr Tiutyk <trofimich@gmail.com>
SPDX-License-Identifier: MIT
License: https://opensource.org/license/mit
*)

(*!
<summary>Provides LIFO insertion and destructive top removal.</summary>
<description>
Successful insertion transfers disposal responsibility for owned payload; borrowed payload must remain alive
while stored. The caller-side descriptor copy is not reset and must not be released again after transfer.
Independent owning aliases and overlapping owned allocations are unsupported. Peek borrows the top; RemoveLast
releases it rather than transferring it to the caller. Clear releases owned payload and dynamic backing
storage.
</description>
*)

INTERFACE IStack EXTENDS IReadOnlyStack

(*!
<summary>Removes all entries and releases dynamic backing storage.</summary>
<description>
Owned payload is released best effort through GENERIC_VALUE.Release; borrowed storage is not freed. Static
capacity and the borrowed validator are retained. Dynamic capacity becomes zero. Returns this collection and
invalidates positions and views. Cleanup callbacks must not reenter mutation.
</description>
*)
METHOD Clear : IStack
END_METHOD

(*!
<summary>Copies a value and appends it to the stack top.</summary>
<description>
Borrows the original during the call. isObject = TRUE requires a live Object FB instance implementing
ICloneable; other data is copied as bytes without recursively cloning references. A prepared copy is released
if insertion fails before acceptance; exceptions propagate. Engine-managed exception objects are unsupported.
The original exception is captured before prepared-copy cleanup, so nested cleanup handling cannot replace
its payload. Terminal OOM takes precedence; capture failure still attempts prepared-copy disposal.
</description>
*)
METHOD PushCopy : IStack
VAR_INPUT
	value : ANY;
	isObject : BOOL := FALSE;
END_VAR
END_METHOD

(*!
<summary>Pushes a descriptor onto the stack top.</summary>
<description>
Successful insertion transfers disposal responsibility for owned payload; borrowed payload must remain alive
while stored. The caller-side descriptor copy is not reset and must not be released again after transfer.
Independent owning aliases and overlapping owned allocations are unsupported. Full static storage raises an
exception. A configured validator is invoked once before any capacity growth or ownership acceptance.
Validation failure leaves the buffer, Length and incoming ownership unchanged; its exception propagates.
Validator callbacks must not mutate this collection.
</description>
*)
METHOD PushGeneric : IStack
VAR_INPUT
	value : TOF_Core.GENERIC_VALUE;
END_VAR
END_METHOD

(*!
<summary>Removes the LIFO top without transferring it to the caller.</summary>
<description>
An empty stack raises CollectionEmptyException. Owned top storage is released best effort, not returned to the
caller. Remaining descriptors are not moved; removal takes constant time apart from payload cleanup. Returns
this stack; positions and views may change. Cleanup callbacks must not reenter mutation.
</description>
*)
METHOD RemoveLast : IStack
END_METHOD

(*!
<summary>Exposes the configured value validator.</summary>
<description>
Borrowed optional reference fixed at initialization. Zero means no validator. The collection does not own or
release it.
</description>
*)
{attribute 'monitoring' := 'call'}
PROPERTY ValueValidator : TOF_Core.IGenericValueValidator
GET
END_GET
END_PROPERTY

END_INTERFACE

// ---- UniqueDataSet/IUniqueDataSet.TcIO
(*!
<summary>Stores unique generic values.</summary>
<description>
SetGeneric replaces a matching entry with the incoming descriptor. SetGeneric preserves disposal
responsibility when the same allocation is reused; transferred caller-side owning aliases must not be released
again. Try lookup/removal operations contain exceptions without rolling back partial effects. Generic query
arguments are borrowed by default. Explicitly requested release in Try operations is attempted even after
lookup failure; caller-side owning aliases are not reset. Lookup uses one equality/hash strategy fixed for the
collection lifetime; zero selects GENERIC_VALUE default equality and hashing. A custom comparer is borrowed,
stays alive and retains stable equality-relevant configuration. Empty descriptors are supported unless
rejected by a validator. No entry or enumeration order is guaranteed; a position is a current storage slot,
not a sorted rank. Do not modify stored descriptors through returned references. Borrowed elements, including
OBJECT instances, stay alive while stored and remain caller-owned. Owned payload must not be deleted through
external aliases. Keep equality/hash-relevant data and comparer configuration stable; remove before changing
them, then insert again. Fields unrelated to equality/hash may change. Callbacks must not mutate elements or
reenter collection mutation. Explicit query release must not dispose of retained storage. Default OBJECT
lookup delegates to Object.Equals/GetHashCode; Clone has its own identity. Discard and populate the index
again after equality-relevant address relocation before further lookup.
</description>
*)
(*
SPDX-FileCopyrightText: © 2026 Oleksandr Tiutyk <trofimich@gmail.com>
SPDX-License-Identifier: MIT
License: https://opensource.org/license/mit
*)

INTERFACE IUniqueDataSet EXTENDS IReadOnlyUniqueDataSet

(*!
<summary>Removes all entries and releases owned payload.</summary>
<description>
Disposal is best effort. Dynamic entry and index storage are released; static capacity and lifetime
comparer/validators are retained. References, positions and active enumeration are invalidated. Cleanup
callbacks must not reenter mutation.
</description>
*)
METHOD Clear : IUniqueDataSet
END_METHOD

(*!
<summary>Removes the entry at a current storage position.</summary>
<description>
The index must be within Length and is not a sorted rank. Removal invalidates positions and references as
entries are compacted; owned payload disposal is best effort. Invalid indices raise an exception.
</description>
*)
METHOD RemoveAt : IUniqueDataSet
VAR_INPUT
	index : DINT;
END_VAR
END_METHOD

(*!
<summary>Copies a value and stores it through SetGeneric.</summary>
<description>
Borrows the original during the call. isObject = TRUE requires a live Object FB instance implementing
ICloneable; other data is copied as bytes without recursively cloning references. A prepared copy is released
if insertion fails before acceptance; exceptions propagate. Engine-managed exception objects are unsupported.
Any index output is meaningful only on success.
The original exception is captured before prepared-copy cleanup, so nested cleanup handling cannot replace
its payload. Terminal OOM takes precedence; capture failure still attempts prepared-copy disposal.
</description>
*)
METHOD SetCopy : IUniqueDataSet
VAR_INPUT
	value : ANY;
	isObject : BOOL := FALSE;
END_VAR
VAR_OUTPUT
	index : DINT;
END_VAR
END_METHOD

(*!
<summary>Inserts a value or replaces the matching entry with the incoming descriptor.</summary>
<description>
Uses the lifetime equality/hash strategy, with no ordering guarantee. Empty descriptors are permitted unless
rejected by a validator. A successful call accepts incoming owned storage; borrowed payload must remain alive
while stored. Validation, lookup and growth precede acceptance; failure before acceptance leaves ownership
with the caller. A displaced owned allocation is released after replacement. Reusing the same allocation does
not release it and preserves existing ownership or accepts incoming ownership, without implicitly returning
ownership to the caller. Caller-side descriptor copies are not reset; transferred owning aliases must not be
released or reused as owners. Aliases must have compatible disposal semantics; overlapping owned ranges and
ownership already held by another entry or owner are not supported. Callbacks must not mutate or reenter this
collection. Cleanup through GENERIC_VALUE.Release is best effort and does not guarantee deallocation. The
index output is valid only on success.
</description>
*)
//!<param name="value">Incoming descriptor; owned storage is transferred on success.</param>
METHOD SetGeneric : IUniqueDataSet
VAR_INPUT
	value : TOF_Core.GENERIC_VALUE;
END_VAR
VAR_OUTPUT
	index : DINT;
END_VAR
END_METHOD

(*!
<summary>Attempts to remove a matching entry.</summary>
<description>
Returns the collection for chaining. removed is TRUE only after the matching entry has been removed; FALSE
means no completed removal was reported. Removal is not transactional and does not prove successful
destruction of an owned payload. Catches exceptions without propagating them or clearing terminal allocation
state. Partial changes are not rolled back. The raw ANY argument is borrowed without cloning or ownership
transfer. isObject = TRUE requires a live Object function-block instance, not a pointer or interface variable.
FALSE uses ordinary runtime type mapping. The caller keeps the query storage alive for the call.
After nested calls and requested cleanup, a fatal allocation state forces the reported outcome to failure.
This does not roll back completed removal or reset the application-wide fatal latch.
</description>
*)
//!<param name="isObject">Explicitly interprets the raw argument as a live Object instance.</param>
METHOD TryRemove : IUniqueDataSet
VAR_INPUT
	value : ANY;
	isObject : BOOL := FALSE;
END_VAR
VAR_OUTPUT
	removed : BOOL;
END_VAR
END_METHOD

(*!
<summary>Attempts to remove a matching entry.</summary>
<description>
Returns the collection for chaining. removed is TRUE only after the matching entry has been removed; FALSE
means no completed removal was reported. Removal is not transactional and does not prove successful
destruction of an owned payload. Catches exceptions without propagating them or clearing terminal allocation
state. Partial changes are not rolled back. The query is borrowed by default. When releaseValue is explicitly
TRUE, attempts to release the supplied generic argument after lookup/removal even on failure. The caller must
have disposal rights and must not reuse aliases of an owned argument after release.
After nested calls and requested cleanup, a fatal allocation state forces the reported outcome to failure.
This does not roll back completed removal or reset the application-wide fatal latch.
</description>
*)
METHOD TryRemoveGeneric : IUniqueDataSet
VAR_INPUT
	value : TOF_Core.GENERIC_VALUE;
	releaseValue : BOOL := FALSE;
END_VAR
VAR_OUTPUT
	removed : BOOL;
END_VAR
END_METHOD

(*!
<summary>Exposes the configured value validator.</summary>
<description>
Borrowed optional reference fixed at initialization. Zero means no validator. The collection does not own or
release it.
</description>
*)
{attribute 'monitoring' := 'call'}
PROPERTY ValueValidator : TOF_Core.IGenericValueValidator
GET
END_GET
END_PROPERTY

END_INTERFACE

// ---- UniqueDataSet/IReadOnlyUniqueDataSet.TcIO
(*
SPDX-FileCopyrightText: © 2026 Oleksandr Tiutyk <trofimich@gmail.com>
SPDX-License-Identifier: MIT
License: https://opensource.org/license/mit
*)

(*!
<summary>Provides lookup and indexed access to a collection of unique generic values.</summary>
<description>
Generic query descriptors are borrowed by default. Explicit release disposes only owned query storage and does
not reset caller-side aliases. The source collection and borrowed payload must remain alive while returned
references are used; mutation can invalidate positions and references. Lookup uses one equality/hash strategy
fixed for the collection lifetime; zero selects GENERIC_VALUE default equality and hashing. A custom comparer
is borrowed, stays alive and retains stable equality-relevant configuration. Empty descriptors are supported
unless rejected by a validator. No entry or enumeration order is guaranteed; a position is a current storage
slot, not a sorted rank. Do not modify stored descriptors through returned references. Borrowed elements,
including OBJECT instances, stay alive while stored and remain caller-owned. Owned payload must not be deleted
through external aliases. Keep equality/hash-relevant data and comparer configuration stable; remove before
changing them, then insert again. Fields unrelated to equality/hash may change. Callbacks must not mutate
elements or reenter collection mutation. Explicit query release must not dispose of retained storage. Default
OBJECT lookup delegates to Object.Equals/GetHashCode; Clone has its own identity. Discard and populate the
index again after equality-relevant address relocation before further lookup.
</description>
*)
INTERFACE IReadOnlyUniqueDataSet EXTENDS ICollection

(*!
<summary>Reports whether a matching raw query exists.</summary>
<description>
The raw ANY argument is borrowed without cloning or ownership transfer. isObject = TRUE requires a live Object
function-block instance, not a pointer or interface variable. FALSE uses ordinary runtime type mapping. The
caller keeps the query storage alive for the call.
</description>
*)
//!<param name="isObject">Explicitly interprets the raw argument as a live Object instance.</param>
METHOD Contains : BOOL
VAR_INPUT
	value : ANY;
	isObject : BOOL := FALSE;
END_VAR
END_METHOD

(*!
<summary>Reports whether a matching entry exists for a borrowed generic query.</summary>
<description>
The query is borrowed by default. Explicit release requests disposal of owned query storage after lookup
completes, including a missing result. Requested release is attempted after both successful lookup and lookup
failure. Before cleanup, the original framework exception is retained and a borrowed static system exception
is cloned to preserve its code, catch point and timestamps across cleanup callbacks. The captured exception is
then propagated through ExceptionManager.Throw in the current cyclic task; native errors use the framework
SystemException representation. If capturing the system exception fails with terminal OOM, query cleanup is
still attempted and terminal OOM takes precedence. Terminal allocation state is never cleared. Release is best
effort and does not prove successful deallocation. Cleanup callbacks must not reenter collection mutation.
Release resets only the local descriptor copy; the caller must have disposal rights and must not reuse or
release owning aliases afterwards. Borrowed payload is not freed.
</description>
*)
METHOD ContainsGeneric : BOOL
VAR_INPUT
	value : TOF_Core.GENERIC_VALUE;
	releaseValue : BOOL := FALSE;
END_VAR
END_METHOD

(*!
<summary>Borrows the entry at a current storage position.</summary>
<description>
The index must be within Length and is not a sorted rank; otherwise an exception is raised. The returned
descriptor reference and payload remain collection-owned or borrowed from their original owner. Do not mutate
the descriptor or dispose of its payload through this view. Mutation or destruction may invalidate the
reference.
</description>
*)
METHOD GetByIndex : REFERENCE TO TOF_Core.GENERIC_VALUE
VAR_INPUT
	index : DINT;
END_VAR
END_METHOD

(*!
<summary>Returns the matching entry position, or a negative value when absent.</summary>
<description>
The query is borrowed by default. Explicit release requests disposal of owned query storage after lookup
completes, including a missing result. Requested release is attempted after both successful lookup and lookup
failure. Before cleanup, the original framework exception is retained and a borrowed static system exception
is cloned to preserve its code, catch point and timestamps across cleanup callbacks. The captured exception is
then propagated through ExceptionManager.Throw in the current cyclic task; native errors use the framework
SystemException representation. If capturing the system exception fails with terminal OOM, query cleanup is
still attempted and terminal OOM takes precedence. Terminal allocation state is never cleared. Release is best
effort and does not prove successful deallocation. Cleanup callbacks must not reenter collection mutation.
Release resets only the local descriptor copy; the caller must have disposal rights and must not reuse or
release owning aliases afterwards. Borrowed payload is not freed. The position is a current storage slot with
no sorted-rank guarantee; mutation may invalidate it.
</description>
*)
METHOD GetGenericValuePosition : DINT
VAR_INPUT
	value : TOF_Core.GENERIC_VALUE;
	releaseValue : BOOL := FALSE;
END_VAR
END_METHOD

(*!
<summary>Returns the matching storage position, or a negative value when absent.</summary>
<description>
The raw ANY argument is borrowed without cloning or ownership transfer. isObject = TRUE requires a live Object
function-block instance, not a pointer or interface variable. FALSE uses ordinary runtime type mapping. The
caller keeps the query storage alive for the call. The position is a current storage slot with no sorted-rank
guarantee; mutation may invalidate it.
</description>
*)
//!<param name="isObject">Explicitly interprets the raw argument as a live Object instance.</param>
METHOD GetValuePosition : DINT
VAR_INPUT
	value : ANY;
	isObject : BOOL := FALSE;
END_VAR
END_METHOD

END_INTERFACE

// ---- ByteList/ByteList.TcPOU
(*
SPDX-FileCopyrightText: © 2026 Oleksandr Tiutyk <trofimich@gmail.com>
SPDX-License-Identifier: MIT
License: https://opensource.org/license/mit
*)

(*!
<summary>Stores a sequence of bytes with fixed or dynamic capacity.</summary>
<description>
CreateEnumerator allocates an independent cursor owned by its caller. The collection must remain alive while
that cursor is used. Static capacity zero selects dynamic storage; otherwise bytes reside in the instance.
DataAddress exposes internal storage: external reassignment invalidates the collection, and growth or
Clear(TRUE) invalidates borrowed addresses. Raw copy methods do not adopt input memory. Remove by value leaves
the collection unchanged when no match exists, including on an empty dynamic instance. WriteData centralizes
capacity checks, writes and buffer replacement. Internal sources and overlapping ranges are supported when the
full source range is readable; growth keeps the old buffer alive until copying completes. Derived callers of
WriteData must satisfy its validated-input preconditions.
Instances cannot be assigned by value: copying backing pointers or disposal responsibility would create
unsafe aliases. Interface references still borrow this instance; copying an interface does not clone storage.
</description>
*)

{attribute 'no_explicit_call' := 'do not call this function block directly'}
FUNCTION_BLOCK ByteList 
VAR_GENERIC CONSTANT
	{attribute 'hide'} 
	//! <summary>Inline capacity; zero selects dynamic backing storage.</summary>
	_StaticCapacity : TOF_Core.DINT_LENGTH := 0;
END_VAR
EXTENDS TOF_Core.Object IMPLEMENTS IByteList
VAR_OUTPUT
	//! <summary>Borrows backing bytes; growth or released capacity invalidates the address.</summary>
	DataAddress : POINTER TO BYTE;
END_VAR
VAR_STAT
	//! <summary>Class name shared by all instances of this function block.</summary>
	{attribute 'hide'} 
	_ClassName : STRING := __POUNAME();
END_VAR
VAR
	{attribute 'hide'} 
	_StaticArray : ARRAY [0.._StaticCapacity - 1] OF BYTE;
	
	{attribute 'hide'} 
	_DynamicCapacity : TOF_Core.DINT_LENGTH;
	{attribute 'hide'} 
	_Length : DINT;
END_VAR

(*!
<summary>Appends the raw storage bytes of an ANY argument.</summary>
<description>
Borrows the argument for copying and uses its full runtime size, including string capacity and structure
padding. Not portable serialization or object cloning. Shares AppendData capacity checks, overlap support and
failure behavior. Descendants cannot override this storage operation; capacity, indexing and disposal remain
governed by this collection implementation.
</description>
*)
METHOD FINAL AppendAny : IByteList
VAR_INPUT
	data : ANY;
END_VAR
AppendAny := AppendData(data := data.pValue, dataSize := TO_DINT(data.diSize));
END_METHOD

(*!
<summary>Appends one byte by value.</summary>
<description>
Returns this list. Full static storage raises an exception; dynamic growth uses checked allocation and
terminal OOM handling. Descendants cannot override this storage operation; capacity, indexing and disposal
remain governed by this collection implementation.
</description>
*)
METHOD FINAL AppendByte : IByteList
VAR_INPUT
	value : BYTE;
END_VAR
AppendByte := AppendData(data := ADR(value), dataSize := 1);
END_METHOD

(*!
<summary>Appends bytes copied from a borrowed memory range.</summary>
<description>
Null data or zero dataSize is a no-op before size validation. Otherwise the source must be readable and
negative sizes or a resulting length outside DINT raise ArgumentOutOfRangeException before copying. Static
capacity exhaustion raises StaticCollectionFullException. Dynamic allocation uses checked growth and terminal
OOM handling. The existing growth increment (free capacity plus input size) is retained and must also fit. The
source may refer to this collection buffer, including overlapping ranges. The caller must provide a readable
range of dataSize bytes; growth keeps the old buffer alive until copying completes. No restriction to logical
Length is imposed on the source. Returns this list. Descendants cannot override this storage operation;
capacity, indexing and disposal remain governed by this collection implementation.
</description>
*)
METHOD FINAL AppendData : IByteList
VAR_INPUT
	data : POINTER TO BYTE;
	dataSize : TOF_Core.DINT_LENGTH;
END_VAR
AppendData := THIS^;

IF data = 0 OR_ELSE dataSize = TOF_Core.SignedInt32.ZERO THEN
	RETURN;
END_IF

IF dataSize < TOF_Core.SignedInt32.ZERO
	OR_ELSE dataSize > TOF_Core.SignedInt32.MAX_VALUE - _Length
THEN
	TOF_Core.Exceptions.ThrowArgumentOutOfRange(
		sourceNamespaceName := NamespaceName,
		sourceClassName := ClassName,
		sourcePOUName := __POUNAME(),
		sourcePosition := __POSITION(),
		argumentName := 'dataSize',
		argumentValue := dataSize
	);
END_IF

WriteData(
	data := data,
	dataSize := dataSize,
	startIndex := _Length,
	requestedCapacity := TO_ULINT(Capacity) + TO_ULINT(Capacity - _Length) + TO_ULINT(dataSize)
);
END_METHOD

(*!
<summary>Appends the raw bytes referenced by a generic descriptor.</summary>
<description>
Borrows the descriptor without adopting or releasing it. Copies Address and Size without value conversion or
object cloning. Size above SignedInt32.MAX_VALUE raises ArgumentOutOfRangeException before narrowing,
including for a null Address. Shares AppendData aliasing and failure behavior. Descendants cannot override
this storage operation; capacity, indexing and disposal remain governed by this collection implementation.
</description>
*)
METHOD FINAL AppendGeneric : IByteList
VAR_INPUT
	data : TOF_Core.GENERIC_VALUE;
END_VAR
IF data.Size > TO_ULINT(TOF_Core.SignedInt32.MAX_VALUE) THEN
	TOF_Core.Exceptions.ThrowArgumentOutOfRange(
		sourceNamespaceName := NamespaceName,
		sourceClassName := ClassName,
		sourcePOUName := __POUNAME(),
		sourcePosition := __POSITION(),
		argumentName := 'data.Size',
		argumentValue := data.Size
	);
END_IF

AppendGeneric := AppendData(data := data.Address, dataSize := TO_DINT(data.Size));
END_METHOD

(*!
<summary>Reports the currently allocated number of slots.</summary>
<description>
Units are bytes for ByteList and entries for other collections. Static capacity is fixed; dynamic capacity can
change on growth or clearing. This is not a guarantee that the next allocation succeeds.
</description>
*)
{attribute 'monitoring' := 'call'}
PROPERTY FINAL Capacity : TOF_Core.DINT_LENGTH
GET
Capacity := SEL(_StaticCapacity = 0, _StaticCapacity, _DynamicCapacity);
END_GET
END_PROPERTY

(*!
<summary>Borrows the concrete collection class name without transferring storage ownership.</summary>
*)
{attribute 'monitoring' := 'call'}
PROPERTY ClassName : REFERENCE TO STRING
GET
ClassName REF= _ClassName;
END_GET
END_PROPERTY

(*!
<summary>Resets the byte count and optionally releases dynamic storage.</summary>
<description>
The default retains capacity for reuse. releaseDynamicMemory = TRUE deletes dynamic storage and sets capacity
to zero. Static storage is retained. Returns this list; old contents are no longer logical entries.
Descendants cannot override this storage operation; capacity, indexing and disposal remain governed by this
collection implementation.
</description>
*)
METHOD FINAL Clear : IByteList
VAR_INPUT
	releaseDynamicMemory : BOOL := FALSE;
END_VAR
Clear := THIS^;

IF releaseDynamicMemory AND_THEN Dynamic AND_THEN _DynamicCapacity > 0 THEN
	__DELETE(DataAddress);
	_DynamicCapacity := 0;
END_IF

_Length := 0;
END_METHOD

(*!
<summary>Creates an independent enumerator owned by the caller.</summary>
<description>
The caller must explicitly release the enumerator and keep this collection alive while using it. Allocation
failure invokes DynamicMemoryManager.RaiseAllocationFailure without a heap exception; it is terminal and is
not returned as a recoverable null result.
</description>
*)
METHOD CreateEnumerator : TOF_Core.IEnumerator
VAR
	enumerator : POINTER TO ByteListEnumerator;
END_VAR
enumerator := __NEW(ByteListEnumerator(list := THIS^));

IF enumerator = 0 THEN
	TOF_Core.DynamicMemoryManager.RaiseAllocationFailure();
END_IF

CreateEnumerator := enumerator^;
END_METHOD

(*!
<summary>Reports whether storage can grow dynamically.</summary>
<description>
Static capacity zero selects dynamic storage. Dynamic collections can still fail to allocate.
</description>
*)
{attribute 'monitoring' := 'call'}
PROPERTY FINAL Dynamic : BOOL
GET
Dynamic := _StaticCapacity = 0;
END_GET
END_PROPERTY

(*!
<summary>Reports whether the collection has no entries.</summary>
<description>
Reflects Length; not a check of payload lifetime or memory health.
</description>
*)
{attribute 'monitoring' := 'call'}
PROPERTY FINAL Empty : BOOL
GET
Empty := _Length <= 0;
END_GET
END_PROPERTY

(*!
<summary>Releases dynamic byte storage during destruction.</summary>
<description>
Calls Clear(releaseDynamicMemory := TRUE); inline storage is not separately deleted. Lifecycle methods must complete without
exceptions. No separate copy-code ownership handoff is implemented.
</description>
*)

METHOD FB_exit : BOOL
VAR_INPUT
	bInCopyCode : BOOL; 
END_VAR
Clear(releaseDynamicMemory := TRUE);
END_METHOD

(*!
<summary>Binds inline byte storage for a static instance.</summary>
<description>
No allocation or callbacks are performed. Dynamic instances start without a backing buffer. No explicit
online-change relocation repair is implemented.
</description>
*)
METHOD FB_init : BOOL
VAR_INPUT
	bInitRetains : BOOL; // TRUE: the retain variables are initialized (reset warm / reset cold)
	bInCopyCode : BOOL; // TRUE: the instance will be copied to the copy code afterward (online change)
END_VAR
IF NOT Dynamic THEN
	DataAddress := ADR(_StaticArray); 
END_IF
END_METHOD

(*!
<summary>Finds the first occurrence of a byte.</summary>
<description>
Searches from zero. TRUE makes index valid; on FALSE no index is promised. The collection is unchanged.
Descendants cannot override this storage operation; capacity, indexing and disposal remain governed by this
collection implementation.
</description>
*)
METHOD FINAL Find : BOOL
VAR_INPUT
	value : BYTE;
END_VAR
VAR_OUTPUT
	index : TOF_Core.DINT_INDEX;
END_VAR
VAR
	i : DINT;	
END_VAR
IF _Length > 0 THEN
	FOR i := 0 TO _Length - 1 DO
		IF DataAddress[i] = value THEN
			index := i;
			Find := TRUE;
			RETURN;
		END_IF 	
	END_FOR
END_IF
END_METHOD

(*!
<summary>Reports whether fixed-capacity storage has no free slot.</summary>
<description>
Dynamic collections report FALSE even when Length equals Capacity. This does not guarantee available heap
memory.
</description>
*)
{attribute 'monitoring' := 'call'}
PROPERTY FINAL Full : BOOL
GET
Full := _StaticCapacity <> 0 AND_THEN _Length >= _StaticCapacity;
END_GET
END_PROPERTY

(*!
<summary>Returns the byte at an existing zero-based position.</summary>
<description>
Raises an exception when backing storage is absent or the index is outside Length. The result is a byte copy.
Descendants cannot override this storage operation; capacity, indexing and disposal remain governed by this
collection implementation.
</description>
*)
METHOD FINAL Get : BYTE
VAR_INPUT
	index : TOF_Core.DINT_INDEX;
END_VAR
IF DataAddress = 0 THEN
	TOF_Core.Exceptions.ThrowStandard(
		sourceNamespaceName := NamespaceName,
		sourceClassName := ClassName,
		sourcePOUName := __POUNAME(),
		sourcePosition := __POSITION(),
		message := "Dynamic byte array is empty"
	);
END_IF

IF index < 0 THEN
	TOF_Core.Exceptions.ThrowStandard(
		sourceNamespaceName := NamespaceName,
		sourceClassName := ClassName,
		sourcePOUName := __POUNAME(),
		sourcePosition := __POSITION(),
		message := "Index is less then zero"
	);
END_IF

IF index >= _Length THEN
	TOF_Core.Exceptions.ThrowStandard(
		sourceNamespaceName := NamespaceName,
		sourceClassName := ClassName,
		sourcePOUName := __POUNAME(),
		sourcePosition := __POSITION(),
		message := "Index is too large"
	);
END_IF

Get := DataAddress[index];
END_METHOD

(*!
<summary>Reports the number of stored entries.</summary>
<description>
Units are bytes for ByteList and entries for other collections. Existing positions range from zero through
Length minus one.
</description>
*)
{attribute 'monitoring' := 'call'}
PROPERTY FINAL Length : TOF_Core.DINT_LENGTH
GET
Length := _Length;
END_GET
END_PROPERTY

(*!
<summary>Loads the full raw representation of an ANY argument at a position.</summary>
<description>
Delegates to LoadFromData using the runtime byte size, including padding and string capacity. Borrows the
source and may truncate the previous tail. Shares LoadFromData limits; not portable serialization. Descendants
cannot override this storage operation; capacity, indexing and disposal remain governed by this collection
implementation.
</description>
*)
METHOD FINAL LoadFromAny : IByteList
VAR_INPUT
	data : ANY;
	startIndex : TOF_Core.DINT_INDEX := 0;
END_VAR
LoadFromAny := LoadFromData(data := data.pValue, dataSize := TO_DINT(data.diSize), startIndex := startIndex);
END_METHOD

(*!
<summary>Copies bytes at a position and sets Length to the end of the copy.</summary>
<description>
startIndex must lie between zero and old Length inclusive, and dataSize must be nonnegative; invalid arguments
raise ArgumentOutOfRangeException. Null data or zero size leaves Length unchanged after these checks. For a
nonempty copy, the resulting length is checked against DINT before arithmetic or mutation. The prefix remains
and the tail beyond the new end is logically truncated. Static capacity exhaustion raises
StaticCollectionFullException; dynamic growth uses checked allocation and terminal OOM handling. Internal
sources and overlapping ranges are supported. The caller must provide a readable source range of dataSize
bytes; the old buffer remains alive throughout copying on growth. No restriction to logical Length is imposed
on the source. Returns this list. Descendants cannot override this storage operation; capacity, indexing and
disposal remain governed by this collection implementation.
</description>
*)
METHOD FINAL LoadFromData : IByteList
VAR_INPUT
	data : POINTER TO BYTE;
	dataSize : TOF_Core.DINT_LENGTH;
	startIndex : TOF_Core.DINT_INDEX := 0;
END_VAR
IF startIndex < TOF_Core.SignedInt32.ZERO OR_ELSE startIndex > _Length THEN
	TOF_Core.Exceptions.ThrowArgumentOutOfRange(
		sourceNamespaceName := NamespaceName,
		sourceClassName := ClassName,
		sourcePOUName := __POUNAME(),
		sourcePosition := __POSITION(),
		argumentName := 'startIndex',
		argumentValue := startIndex
	);
END_IF

IF dataSize < TOF_Core.SignedInt32.ZERO THEN
	TOF_Core.Exceptions.ThrowArgumentOutOfRange(
		sourceNamespaceName := NamespaceName,
		sourceClassName := ClassName,
		sourcePOUName := __POUNAME(),
		sourcePosition := __POSITION(),
		argumentName := 'dataSize',
		argumentValue := dataSize
	);
END_IF

LoadFromData := THIS^;
 
IF data = 0 OR_ELSE dataSize = TOF_Core.SignedInt32.ZERO THEN
	RETURN;
END_IF

IF dataSize > TOF_Core.SignedInt32.MAX_VALUE - startIndex THEN
	TOF_Core.Exceptions.ThrowArgumentOutOfRange(
		sourceNamespaceName := NamespaceName,
		sourceClassName := ClassName,
		sourcePOUName := __POUNAME(),
		sourcePosition := __POSITION(),
		argumentName := 'dataSize',
		argumentValue := dataSize
	);
END_IF

WriteData(
		data := data,
		dataSize := dataSize,
		startIndex := startIndex,
		requestedCapacity := TO_ULINT(startIndex) + TO_ULINT(dataSize)
	);
END_METHOD

(*!
<summary>Loads the byte range referenced by a generic descriptor.</summary>
<description>
Borrows the descriptor without adoption or release. Size above SignedInt32.MAX_VALUE raises
ArgumentOutOfRangeException before narrowing, including for a null Address. Shares LoadFromData index checks,
truncation, aliasing and failure behavior. Descendants cannot override this storage operation; capacity,
indexing and disposal remain governed by this collection implementation.
</description>
*)
METHOD FINAL LoadFromGeneric : IByteList
VAR_INPUT
	data : TOF_Core.GENERIC_VALUE;
	startIndex : TOF_Core.DINT_INDEX := 0;
END_VAR
IF data.Size > TO_ULINT(TOF_Core.SignedInt32.MAX_VALUE) THEN
	TOF_Core.Exceptions.ThrowArgumentOutOfRange(
		sourceNamespaceName := NamespaceName,
		sourceClassName := ClassName,
		sourcePOUName := __POUNAME(),
		sourcePosition := __POSITION(),
		argumentName := 'data.Size',
		argumentValue := data.Size
	);
END_IF

LoadFromGeneric := LoadFromData(data := data.Address, dataSize := TO_DINT(data.Size), startIndex := startIndex);
END_METHOD

(*!
<summary>Provides the library namespace for diagnostics.</summary>
<description>
Borrowed read-only reference to compiler-initialized metadata; no ownership transfer.
</description>
*)
{attribute 'monitoring' := 'call'}
PROPERTY NamespaceName : REFERENCE TO STRING
GET
NamespaceName REF= CurrentNamespace.Name;
END_GET
END_PROPERTY

(*!
<summary>Removes the first occurrence of a byte if present.</summary>
<description>
Removes only the first matching byte, compacts later bytes through RemoveAt and returns this list. An absent
value or an empty static or dynamic list leaves the collection unchanged without raising an exception for
absence. Capacity is retained. Requires an intact collection whose backing storage remains valid for its
logical contents. Descendants cannot override this storage operation; capacity, indexing and disposal remain
governed by this collection implementation.
</description>
*)
METHOD FINAL Remove : IByteList
VAR_INPUT
	value : BYTE;
END_VAR
VAR
	index : DINT;
END_VAR
Remove := THIS^;

IF Find(value := value, index => index) THEN
	RemoveAt(index := index, count := 1);
END_IF
END_METHOD

(*!
<summary>Removes a contiguous byte range and compacts remaining bytes.</summary>
<description>
Requires an existing index and a nonnegative count no greater than the remaining length; otherwise raises
ArgumentOutOfRangeException. The range is checked by subtraction before computing its end. Zero count is a
no-op only after index validation. Capacity is retained. Returns this list. Descendants cannot override this
storage operation; capacity, indexing and disposal remain governed by this collection implementation.
</description>
*)
METHOD FINAL RemoveAt : IByteList
VAR_INPUT
	index : TOF_Core.DINT_INDEX;
	count : TOF_Core.DINT_LENGTH := 1;
END_VAR
IF index < TOF_Core.SignedInt32.ZERO OR_ELSE index >= _Length THEN
	TOF_Core.Exceptions.ThrowArgumentOutOfRange(
		sourceNamespaceName := NamespaceName,
		sourceClassName := ClassName,
		sourcePOUName := __POUNAME(),
		sourcePosition := __POSITION(),
		argumentName := 'index',
		argumentValue := index
	);
END_IF

IF count < TOF_Core.SignedInt32.ZERO OR_ELSE count > _Length - index THEN
	TOF_Core.Exceptions.ThrowArgumentOutOfRange(
		sourceNamespaceName := NamespaceName,
		sourceClassName := ClassName,
		sourcePOUName := __POUNAME(),
		sourcePosition := __POSITION(),
		argumentName := 'count',
		argumentValue := count
	);
END_IF

RemoveAt := THIS^;

IF count = TOF_Core.SignedInt32.ZERO THEN
	RETURN;
END_IF

IF count <> _Length THEN
	Tc2_System.MEMMOVE(
		destAddr := DataAddress + TO_LWORD(index),
		srcAddr := DataAddress + TO_LWORD(index + count),
		n := TO_UDINT(_Length - index - count)
	);
END_IF

_Length := _Length - count;
END_METHOD

(*!
<summary>Reports the size of this function-block instance.</summary>
<description>
Measured in bytes; includes inline storage but excludes separately allocated buffers, payload and enumerators.
</description>
*)
{attribute 'monitoring' := 'call'}
PROPERTY SelfSize : ULINT
GET
SelfSize := XSIZEOF(THIS^);
END_GET
END_PROPERTY

(*!
<summary>Overwrites one existing byte.</summary>
<description>
Requires allocated storage and an index within Length; otherwise raises an exception. Length and Capacity are
unchanged. Returns this list. Descendants cannot override this storage operation; capacity, indexing and
disposal remain governed by this collection implementation.
</description>
*)
METHOD FINAL Set : IByteList
VAR_INPUT
	index : TOF_Core.DINT_INDEX;
	value : BYTE;
END_VAR
IF DataAddress = 0 THEN
	TOF_Core.Exceptions.ThrowStandard(
		sourceNamespaceName := NamespaceName,
		sourceClassName := ClassName,
		sourcePOUName := __POUNAME(),
		sourcePosition := __POSITION(),
		message := "Dynamic byte array is empty"
	);
END_IF

IF index < 0 THEN
	TOF_Core.Exceptions.ThrowStandard(
		sourceNamespaceName := NamespaceName,
		sourceClassName := ClassName,
		sourcePOUName := __POUNAME(),
		sourcePosition := __POSITION(),
		message := "Index is less then zero"
	);
END_IF

IF index >= _Length THEN
	TOF_Core.Exceptions.ThrowStandard(
		sourceNamespaceName := NamespaceName,
		sourceClassName := ClassName,
		sourcePOUName := __POUNAME(),
		sourcePosition := __POSITION(),
		message := "Index is too large"
	);
END_IF

Set := THIS^;

DataAddress[index] := value;
END_METHOD

(*!
<summary>Writes a prepared byte range and centrally manages any buffer replacement.</summary>
<description>
The caller must validate a non-null readable source, positive dataSize, startIndex within Length and a
representable resulting length. requestedCapacity specifies the growth policy and is used only when the write
exceeds Capacity. It must cover the resulting length and fit DINT. Static exhaustion raises
StaticCollectionFullException. Invalid growth capacity raises ArgumentOutOfRangeException. Null NEW invokes
terminal allocation failure before mutation. Without growth, MEMMOVE supports overlapping ranges. With growth,
the old buffer remains alive until both existing bytes and source bytes have been copied; only then are
pointer, capacity and length committed and the old allocation deleted. Source ranges may include the
collection buffer, provided the full range is readable; no restriction to logical Length is imposed. Borrowed
buffer addresses are invalidated by growth. This helper does not validate arbitrary pointer lifetime.
</description>
*)
METHOD PROTECTED FINAL WriteData
VAR_INPUT
	data : POINTER TO BYTE;
	dataSize : TOF_Core.DINT_LENGTH;
	startIndex : TOF_Core.DINT_INDEX;
	requestedCapacity : ULINT;
END_VAR
VAR
	newLength : DINT;
	newMemory : POINTER TO BYTE;
	oldMemory : POINTER TO BYTE;

END_VAR
newLength := startIndex + dataSize;

IF newLength <= Capacity THEN
	Tc2_System.MEMMOVE(destAddr := DataAddress + TO_DWORD(startIndex), srcAddr := data, n := TO_UDINT(dataSize));
	_Length := newLength;
	RETURN;
END_IF

IF NOT Dynamic THEN
	TOF_Core.Exceptions.ThrowStaticCollectionFull(
		sourceNamespaceName := NamespaceName,
		sourceClassName := ClassName,
		sourcePOUName := __POUNAME(),
		sourcePosition := __POSITION(),
		collectionName := GetName(),
		capacity := TO_UDINT(Capacity)
	);
END_IF

IF requestedCapacity < TO_ULINT(newLength)
	OR_ELSE requestedCapacity > TO_ULINT(TOF_Core.SignedInt32.MAX_VALUE)
THEN
	TOF_Core.Exceptions.ThrowArgumentOutOfRange(
		sourceNamespaceName := NamespaceName,
		sourceClassName := ClassName,
		sourcePOUName := __POUNAME(),
		sourcePosition := __POSITION(),
		argumentName := 'capacity',
		argumentValue := requestedCapacity
	);
END_IF

newMemory := __NEW(BYTE, TO_UDINT(requestedCapacity));

IF newMemory = 0 THEN
	TOF_Core.DynamicMemoryManager.RaiseAllocationFailure();
END_IF

oldMemory := DataAddress;

IF _Length > TOF_Core.SignedInt32.ZERO THEN
	Tc2_System.MEMCPY(destAddr := newMemory, srcAddr := oldMemory, n := TO_UDINT(_Length));
END_IF

// The source may refer to the old buffer, which remains alive until this copy completes.
Tc2_System.MEMCPY(destAddr := newMemory + TO_DWORD(startIndex), srcAddr := data, n := TO_UDINT(dataSize));

DataAddress := newMemory;
_DynamicCapacity := TO_DINT(requestedCapacity);
_Length := newLength;

IF oldMemory <> 0 THEN
	__DELETE(oldMemory);
END_IF
END_METHOD

END_FUNCTION_BLOCK

// ---- ByteList/ByteListEnumerator.TcPOU
(*
SPDX-FileCopyrightText: © 2026 Oleksandr Tiutyk <trofimich@gmail.com>
SPDX-License-Identifier: MIT
License: https://opensource.org/license/mit
*)

(*!
<summary>Enumerates a borrowed collection using an independent cursor.</summary>
<description>
The source must be non-null, outlive the cursor and remain structurally unchanged during traversal. The caller
explicitly releases a dynamically created cursor. Current borrows a byte cached in this cursor, not the source
buffer; it never transfers ownership. MoveNext stops advancing at the end position of an unchanged source;
repeated exhausted calls return FALSE until Reset.
A null constructor source is diagnosed by traversal/current access, never by FB_init.
</description>
*)

{attribute 'no_explicit_call' := 'do not call this function block directly'}
{attribute 'enable_dynamic_creation'}
FUNCTION_BLOCK ByteListEnumerator EXTENDS TOF_Core.Object IMPLEMENTS TOF_Core.IEnumerator
VAR_STAT
	//! <summary>Class name shared by all instances of this function block.</summary>
	{attribute 'hide'} 
	_ClassName : STRING := __POUNAME();
END_VAR
VAR
	{attribute 'hide'} 
	_List : IReadOnlyByteList;
	{attribute 'hide'} 
	_CurrentIndex : DINT := -1;
	
	{attribute 'hide'} 
	_CurrentByte : BYTE;
	{attribute 'hide'} 
	_GenericValue : TOF_Core.GENERIC_VALUE;	
END_VAR

(*!
<summary>Borrows the concrete cursor class name without transferring storage ownership.</summary>
*)
{attribute 'monitoring' := 'call'}
PROPERTY ClassName : REFERENCE TO STRING
GET
ClassName REF= _ClassName;
END_GET
END_PROPERTY

(*!
<summary>Exposes a read-only borrowed view of the current entry.</summary>
<description>
Reading Current before the first successful MoveNext, after Reset or after exhaustion yields an empty
descriptor. At a valid position, the source byte is copied into cursor-local storage and the returned
descriptor borrows that storage, including when the byte value is zero. Do not modify or release the
descriptor. Keep the cursor alive while using the view; subsequent Current access can overwrite its cached
byte. Cursor movement or reset invalidates the previous view contract.
Missing source raises DataMemberNotSpecifiedException before source access or cursor advancement.
</description>
*)
{attribute 'monitoring' := 'call'}
PROPERTY FINAL Current : REFERENCE TO TOF_Core.GENERIC_VALUE
GET
requireSource();

IF _CurrentIndex >= 0 AND_THEN _CurrentIndex < _List.Length THEN
	_CurrentByte := _List.Get(index := _CurrentIndex); 
	_GenericValue := TOF_Core.GenericValueFactory.FromParts(
		genericTypeClass := TOF_Core.GENERIC_TYPE_CLASS.UINT_8,
		address := ADR(_CurrentByte),
		size := 1,
		memoryManagementBehavior := TOF_Core.GENERIC_MEMORY_MANAGEMENT_BEHAVIOR.STORE_ORIGINAL_REFERENCE_AND_NOT_OWNS_MEMORY
	);
ELSE
	_GenericValue.Reset();
END_IF 

Current REF= _GenericValue;
END_GET
END_PROPERTY

(*!
<summary>Returns the current entry in its concrete representation.</summary>
<description>
Use only after MoveNext returns TRUE and before the next cursor or source change. No result is promised
outside a valid position. The byte is returned by value.
Missing source raises DataMemberNotSpecifiedException before source access or cursor advancement.
</description>
*)
{attribute 'monitoring' := 'call'}
PROPERTY FINAL CurrentByte : BYTE
GET
requireSource();

IF _CurrentIndex >= 0 AND_THEN _CurrentIndex < _List.Length THEN
	CurrentByte := _List.Get(index := _CurrentIndex); 
END_IF
END_GET
END_PROPERTY

(*!
<summary>Binds the borrowed source for enumeration.</summary>
<description>
The source must be non-null and outlive the cursor. Only the reference is assigned; no allocation, callbacks
or throwing validation are performed. A null source remains invalid configuration and is reported by
MoveNext or current-value access without throwing from initialization.
</description>
*)
METHOD FB_init : BOOL
VAR_INPUT
	bInitRetains : BOOL; // TRUE: the retain variables are initialized (reset warm / reset cold)
	bInCopyCode : BOOL;  // TRUE: the instance will be copied to the copy code afterward (online change)
	list : IReadOnlyByteList;
END_VAR
_List := list;
END_METHOD

